// TwinCAT 3 PLC project Untitled1
// ProgramVersion: 3.1.4024.0
// libraries:
//   Tc2_Standard, * (Beckhoff Automation GmbH)
//   Tc2_System, * (Beckhoff Automation GmbH)
//   Tc2_Utilities, * (Beckhoff Automation GmbH)
//   Tc3_Module, * (Beckhoff Automation GmbH)
// project tree:
//   / PlcTask.TcTTO
//   Lib/Any/ ToAnyType.TcPOU (not stored)
//   Lib/ MAIN.TcPOU (not stored)
//   Lib/PrimitiveValues/ ValueLrealRead.TcPOU (not stored), ValueLreal.TcPOU, ValueByte.TcPOU (not stored), ValueByteRead.TcPOU (not stored), ValueDate.TcPOU (not stored), ValueDateRead.TcPOU, ValueDint.TcPOU (not stored), ValueDintRead.TcPOU (not stored), ValueDt.TcPOU (not stored), ValueDtRead.TcPOU (not stored), ValueDword.TcPOU (not stored), ValueDwordRead.TcPOU (not stored), ValueInt.TcPOU, ValueIntRead.TcPOU (not stored), ValueLint.TcPOU, ValueLintRead.TcPOU, ValueLtime.TcPOU (not stored), ValueLtimeRead.TcPOU, ValueLword.TcPOU (not stored), ValueLwordRead.TcPOU (not stored), ValueReal.TcPOU (not stored), ValueRealRead.TcPOU, ValueSint.TcPOU (not stored), ValueSintRead.TcPOU, ValueString.TcPOU, ValueStringRead.TcPOU (not stored), ValueTime.TcPOU (not stored), ValueTimeRead.TcPOU (not stored), ValueTod.TcPOU, ValueTodRead.TcPOU (not stored), ValueUdint.TcPOU (not stored), ValueUdintRead.TcPOU, ValueUint.TcPOU (not stored), ValueUintRead.TcPOU (not stored), ValueUlint.TcPOU, ValueUlintRead.TcPOU, ValueUsint.TcPOU (not stored), ValueUsintRead.TcPOU (not stored), ValueWord.TcPOU (not stored), ValueWordRead.TcPOU (not stored), ValueWstring.TcPOU, ValueWstringRead.TcPOU (not stored)
//   Lib/Startable/ CommandStatus.TcIO (not stored), Startable.TcIO
//   Lib/Value/ Value.TcIO, ValueBase.TcPOU, ValueWithType.TcIO, ValueRead.TcIO (not stored), ValueType.TcDUT
//   Lib/Conversion/ ConvertAnyType.TcPOU (not stored)
// real-time tasks:
//   TASK PlcTask: cycle T#10ms, priority 20, ADS port 350

CONFIGURATION Untitled1
    RESOURCE PLC ON TwinCAT3
        TASK PlcTask(INTERVAL := T#10ms, PRIORITY := 20);
        PROGRAM MAIN WITH PlcTask : MAIN;
    END_RESOURCE
END_CONFIGURATION

// ---- Lib/Value/ValueType.TcDUT
TYPE ValueType : __SYSTEM.TYPE_CLASS; END_TYPE

// ---- Lib/Startable/Startable.TcIO
{attribute 'linkalways'}
INTERFACE Startable EXTENDS __SYSTEM.IQueryInterface

METHOD Start : CommandStatus
END_METHOD

END_INTERFACE

// ---- Lib/Value/Value.TcIO
{attribute 'linkalways'}
INTERFACE Value EXTENDS ValueRead

METHOD Set : BOOL
VAR_INPUT
	source : ANY;
END_VAR
END_METHOD

METHOD SetFromString : BOOL
VAR_INPUT
	value : T_MaxString;
END_VAR
END_METHOD

METHOD SetFromType : BOOL
VAR_INPUT
	source : __SYSTEM.AnyType;
END_VAR
END_METHOD

END_INTERFACE

// ---- Lib/Value/ValueWithType.TcIO
INTERFACE ValueWithType EXTENDS __SYSTEM.IQueryInterface

{attribute 'monitoring' := 'call'}
PROPERTY ValueType : ValueType
GET
END_GET
END_PROPERTY

END_INTERFACE

// ---- Lib/PrimitiveValues/ValueLreal.TcPOU
{attribute 'linkalways'}
{attribute 'hide_all_locals'}
FUNCTION_BLOCK ValueLreal EXTENDS ValueLrealRead IMPLEMENTS Value
VAR
END_VAR

METHOD Set : BOOL
VAR_INPUT
	source : ANY;
END_VAR
Set := ConvertAnyType(source, thisAnyType);
END_METHOD

METHOD SetFromString : BOOL
VAR_INPUT
	value : T_MaxString;
END_VAR
thisValue := STRING_TO_LREAL(value);

SetFromString := TRUE;
END_METHOD

METHOD SetFromType : BOOL
VAR_INPUT
	source : __SYSTEM.AnyType;
END_VAR
SetFromType := ConvertAnyType(source, thisAnyType);
END_METHOD

END_FUNCTION_BLOCK

// ---- Lib/Value/ValueBase.TcPOU
{attribute 'linkalways'}
{attribute 'hide_all_locals'}
FUNCTION_BLOCK ABSTRACT ValueBase IMPLEMENTS ValueWithType
VAR
	_ValueType : ValueType;
	thisAnyType : __SYSTEM.AnyType;
END_VAR

{attribute 'call_after_global_init_slot' := '1'}
{attribute 'call_after_online_change_slot' := '1'}
METHOD PROTECTED ABSTRACT GetThisAnyType
VAR_INPUT
END_VAR
END_METHOD

{attribute 'monitoring' := 'call'}
PROPERTY ValueType : ValueType
GET
ValueType := _ValueType;
END_GET
END_PROPERTY

END_FUNCTION_BLOCK

// ---- Lib/PrimitiveValues/ValueDateRead.TcPOU
{attribute 'linkalways'}
{attribute 'hide_all_locals'}
FUNCTION_BLOCK ValueDateRead EXTENDS ValueBase IMPLEMENTS ValueRead
VAR
	thisValue : DATE;
END_VAR

{attribute 'call_after_global_init_slot' := '1'}
{attribute 'call_after_online_change_slot' := '1'}
METHOD PROTECTED GetThisAnyType
VAR_INPUT
END_VAR
thisAnyType := ToAnyType(thisValue);
END_METHOD

METHOD GetAsType : BOOL
VAR_INPUT
	destination : __SYSTEM.AnyType;
END_VAR
GetAsType := ConvertAnyType(thisAnyType, destination);
END_METHOD

METHOD GetAsString : T_MaxString
VAR_INPUT
END_VAR
GetAsString := DATE_TO_STRING(thisValue);
END_METHOD

METHOD Get : BOOL
VAR_INPUT
	destination : ANY;
END_VAR
Get := ConvertAnyType(thisAnyType, destination);
END_METHOD

METHOD FB_init : BOOL
VAR_INPUT
	bInitRetains : BOOL; // if TRUE, the retain variables are initialized (warm start / cold start)
	bInCopyCode : BOOL;  // if TRUE, the instance afterwards gets moved into the copy code (online change)
END_VAR
_ValueType := __SYSTEM.TYPE_CLASS.TYPE_DATE;
END_METHOD

{attribute 'monitoring' := 'call'}
PROPERTY Value : DATE
GET
Value := thisValue;
END_GET
END_PROPERTY

END_FUNCTION_BLOCK

// ---- Lib/PrimitiveValues/ValueInt.TcPOU
{attribute 'linkalways'}
{attribute 'hide_all_locals'}
FUNCTION_BLOCK ValueInt EXTENDS ValueIntRead IMPLEMENTS Value
VAR
END_VAR

METHOD SetFromType : BOOL
VAR_INPUT
	source : __SYSTEM.AnyType;
END_VAR
SetFromType := ConvertAnyType(source, thisAnyType);
END_METHOD

METHOD SetFromString : BOOL
VAR_INPUT
	value : T_MaxString;
END_VAR
thisValue := STRING_TO_INT(value);

SetFromString := TRUE;
END_METHOD

METHOD Set : BOOL
VAR_INPUT
	source : ANY;
END_VAR
Set := ConvertAnyType(source, thisAnyType);
END_METHOD

END_FUNCTION_BLOCK

// ---- Lib/PrimitiveValues/ValueLint.TcPOU
{attribute 'linkalways'}
{attribute 'hide_all_locals'}
FUNCTION_BLOCK ValueLint EXTENDS ValueLintRead IMPLEMENTS Value
VAR
END_VAR

METHOD SetFromType : BOOL
VAR_INPUT
	source : __SYSTEM.AnyType;
END_VAR
SetFromType := ConvertAnyType(source, thisAnyType);
END_METHOD

METHOD SetFromString : BOOL
VAR_INPUT
	value : T_MaxString;
END_VAR
thisValue := STRING_TO_LINT(value);

SetFromString := TRUE;
END_METHOD

METHOD Set : BOOL
VAR_INPUT
	source : ANY;
END_VAR
Set := ConvertAnyType(source, thisAnyType);
END_METHOD

END_FUNCTION_BLOCK

// ---- Lib/PrimitiveValues/ValueLintRead.TcPOU
{attribute 'linkalways'}
{attribute 'hide_all_locals'}
FUNCTION_BLOCK ValueLintRead EXTENDS ValueBase IMPLEMENTS ValueRead
VAR
	thisValue : LINT;
END_VAR

{attribute 'call_after_global_init_slot' := '1'}
{attribute 'call_after_online_change_slot' := '1'}
METHOD PROTECTED GetThisAnyType
VAR_INPUT
END_VAR
thisAnyType := ToAnyType(thisValue);
END_METHOD

METHOD GetAsType : BOOL
VAR_INPUT
	destination : __SYSTEM.AnyType;
END_VAR
GetAsType := ConvertAnyType(thisAnyType, destination);
END_METHOD

METHOD GetAsString : T_MaxString
VAR_INPUT
END_VAR
GetAsString := TO_STRING(thisValue);
END_METHOD

METHOD Get : BOOL
VAR_INPUT
	destination : ANY;
END_VAR
Get := ConvertAnyType(thisAnyType, destination);
END_METHOD

METHOD FB_init : BOOL
VAR_INPUT
	bInitRetains : BOOL; // if TRUE, the retain variables are initialized (warm start / cold start)
	bInCopyCode : BOOL;  // if TRUE, the instance afterwards gets moved into the copy code (online change)
END_VAR
_ValueType := __SYSTEM.TYPE_CLASS.TYPE_LINT;
END_METHOD

{attribute 'monitoring' := 'call'}
PROPERTY Value : LINT
GET
Value := thisValue;
END_GET
END_PROPERTY

END_FUNCTION_BLOCK

// ---- Lib/PrimitiveValues/ValueLtimeRead.TcPOU
{attribute 'linkalways'}
{attribute 'hide_all_locals'}
FUNCTION_BLOCK ValueLtimeRead EXTENDS ValueBase IMPLEMENTS ValueRead
VAR
	thisValue : LTIME;
END_VAR

{attribute 'call_after_global_init_slot' := '1'}
{attribute 'call_after_online_change_slot' := '1'}
METHOD PROTECTED GetThisAnyType
VAR_INPUT
END_VAR
thisAnyType := ToAnyType(thisValue);
END_METHOD

METHOD GetAsType : BOOL
VAR_INPUT
	destination : __SYSTEM.AnyType;
END_VAR
GetAsType := ConvertAnyType(thisAnyType, destination);
END_METHOD

METHOD GetAsString : T_MaxString
VAR_INPUT
END_VAR
GetAsString := LTIME_TO_STRING(thisValue);
END_METHOD

METHOD Get : BOOL
VAR_INPUT
	destination : ANY;
END_VAR
Get := ConvertAnyType(thisAnyType, destination);
END_METHOD

METHOD FB_init : BOOL
VAR_INPUT
	bInitRetains : BOOL; // if TRUE, the retain variables are initialized (warm start / cold start)
	bInCopyCode : BOOL;  // if TRUE, the instance afterwards gets moved into the copy code (online change)
END_VAR
_ValueType := __SYSTEM.TYPE_CLASS.TYPE_LTIME;
END_METHOD

{attribute 'monitoring' := 'call'}
PROPERTY Value : LTIME
GET
Value := thisValue;
END_GET
END_PROPERTY

END_FUNCTION_BLOCK

// ---- Lib/PrimitiveValues/ValueRealRead.TcPOU
{attribute 'linkalways'}
{attribute 'hide_all_locals'}
FUNCTION_BLOCK ValueRealRead EXTENDS ValueBase IMPLEMENTS ValueRead
VAR
	thisValue : REAL;
END_VAR

{attribute 'call_after_global_init_slot' := '1'}
{attribute 'call_after_online_change_slot' := '1'}
METHOD PROTECTED GetThisAnyType
VAR_INPUT
END_VAR
thisAnyType := ToAnyType(thisValue);
END_METHOD

METHOD GetAsType : BOOL
VAR_INPUT
	destination : __SYSTEM.AnyType;
END_VAR
GetAsType := ConvertAnyType(thisAnyType, destination);
END_METHOD

METHOD GetAsString : T_MaxString
VAR_INPUT
END_VAR
GetAsString := TO_STRING(thisValue);
END_METHOD

METHOD Get : BOOL
VAR_INPUT
	destination : ANY;
END_VAR
Get := ConvertAnyType(thisAnyType, destination);
END_METHOD

METHOD FB_init : BOOL
VAR_INPUT
	bInitRetains : BOOL; // if TRUE, the retain variables are initialized (warm start / cold start)
	bInCopyCode : BOOL;  // if TRUE, the instance afterwards gets moved into the copy code (online change)
END_VAR
_ValueType := __SYSTEM.TYPE_CLASS.TYPE_REAL;
END_METHOD

{attribute 'monitoring' := 'call'}
PROPERTY Value : REAL
GET
Value := thisValue;
END_GET
END_PROPERTY

END_FUNCTION_BLOCK

// ---- Lib/PrimitiveValues/ValueSintRead.TcPOU
{attribute 'linkalways'}
{attribute 'hide_all_locals'}
FUNCTION_BLOCK ValueSintRead EXTENDS ValueBase IMPLEMENTS ValueRead
VAR
	thisValue : SINT;
END_VAR

{attribute 'call_after_global_init_slot' := '1'}
{attribute 'call_after_online_change_slot' := '1'}
METHOD PROTECTED GetThisAnyType
VAR_INPUT
END_VAR
thisAnyType := ToAnyType(thisValue);
END_METHOD

METHOD GetAsType : BOOL
VAR_INPUT
	destination : __SYSTEM.AnyType;
END_VAR
GetAsType := ConvertAnyType(thisAnyType, destination);
END_METHOD

METHOD GetAsString : T_MaxString
VAR_INPUT
END_VAR
GetAsString := TO_STRING(thisValue);
END_METHOD

METHOD Get : BOOL
VAR_INPUT
	destination : ANY;
END_VAR
Get := ConvertAnyType(thisAnyType, destination);
END_METHOD

METHOD FB_init : BOOL
VAR_INPUT
	bInitRetains : BOOL; // if TRUE, the retain variables are initialized (warm start / cold start)
	bInCopyCode : BOOL;  // if TRUE, the instance afterwards gets moved into the copy code (online change)
END_VAR
_ValueType := __SYSTEM.TYPE_CLASS.TYPE_SINT;
END_METHOD

{attribute 'monitoring' := 'call'}
PROPERTY Value : SINT
GET
Value := thisValue;
END_GET
END_PROPERTY

END_FUNCTION_BLOCK

// ---- Lib/PrimitiveValues/ValueString.TcPOU
{attribute 'linkalways'}
{attribute 'hide_all_locals'}
FUNCTION_BLOCK ValueString EXTENDS ValueStringRead IMPLEMENTS Value
VAR
END_VAR

METHOD SetFromType : BOOL
VAR_INPUT
	source : __SYSTEM.AnyType;
END_VAR
SetFromType := ConvertAnyType(source, thisAnyType);
END_METHOD

METHOD SetFromString : BOOL
VAR_INPUT
	value : T_MaxString;
END_VAR
thisValue := value;

SetFromString := TRUE;
END_METHOD

METHOD Set : BOOL
VAR_INPUT
	source : ANY;
END_VAR
Set := ConvertAnyType(source, thisAnyType);
END_METHOD

END_FUNCTION_BLOCK

// ---- Lib/PrimitiveValues/ValueTod.TcPOU
{attribute 'linkalways'}
{attribute 'hide_all_locals'}
FUNCTION_BLOCK ValueTod EXTENDS ValueTodRead IMPLEMENTS Value
VAR
END_VAR

METHOD SetFromType : BOOL
VAR_INPUT
	source : __SYSTEM.AnyType;
END_VAR
SetFromType := ConvertAnyType(source, thisAnyType);
END_METHOD

METHOD SetFromString : BOOL
VAR_INPUT
	value : T_MaxString;
END_VAR
thisValue := STRING_TO_TOD(value);

SetFromString := TRUE;
END_METHOD

METHOD Set : BOOL
VAR_INPUT
	source : ANY;
END_VAR
Set := ConvertAnyType(source, thisAnyType);
END_METHOD

END_FUNCTION_BLOCK

// ---- Lib/PrimitiveValues/ValueUdintRead.TcPOU
{attribute 'linkalways'}
{attribute 'hide_all_locals'}
FUNCTION_BLOCK ValueUdintRead EXTENDS ValueBase IMPLEMENTS ValueRead
VAR
	thisValue : UDINT;
END_VAR

{attribute 'call_after_global_init_slot' := '1'}
{attribute 'call_after_online_change_slot' := '1'}
METHOD PROTECTED GetThisAnyType
VAR_INPUT
END_VAR
thisAnyType := ToAnyType(thisValue);
END_METHOD

METHOD GetAsType : BOOL
VAR_INPUT
	destination : __SYSTEM.AnyType;
END_VAR
GetAsType := ConvertAnyType(thisAnyType, destination);
END_METHOD

METHOD GetAsString : T_MaxString
VAR_INPUT
END_VAR
GetAsString := TO_STRING(thisValue);
END_METHOD

METHOD Get : BOOL
VAR_INPUT
	destination : ANY;
END_VAR
Get := ConvertAnyType(thisAnyType, destination);
END_METHOD

METHOD FB_init : BOOL
VAR_INPUT
	bInitRetains : BOOL; // if TRUE, the retain variables are initialized (warm start / cold start)
	bInCopyCode : BOOL;  // if TRUE, the instance afterwards gets moved into the copy code (online change)
END_VAR
_ValueType := __SYSTEM.TYPE_CLASS.TYPE_UDINT;
END_METHOD

{attribute 'monitoring' := 'call'}
PROPERTY Value : UDINT
GET
Value := thisValue;
END_GET
END_PROPERTY

END_FUNCTION_BLOCK

// ---- Lib/PrimitiveValues/ValueUlint.TcPOU
{attribute 'linkalways'}
{attribute 'hide_all_locals'}
FUNCTION_BLOCK ValueUlint EXTENDS ValueUlintRead IMPLEMENTS Value
VAR
END_VAR

METHOD SetFromType : BOOL
VAR_INPUT
	source : __SYSTEM.AnyType;
END_VAR
SetFromType := ConvertAnyType(source, thisAnyType);
END_METHOD

METHOD SetFromString : BOOL
VAR_INPUT
	value : T_MaxString;
END_VAR
thisValue := STRING_TO_ULINT(value);

SetFromString := TRUE;
END_METHOD

METHOD Set : BOOL
VAR_INPUT
	source : ANY;
END_VAR
Set := ConvertAnyType(source, thisAnyType);
END_METHOD

END_FUNCTION_BLOCK

// ---- Lib/PrimitiveValues/ValueUlintRead.TcPOU
{attribute 'linkalways'}
{attribute 'hide_all_locals'}
FUNCTION_BLOCK ValueUlintRead EXTENDS ValueBase IMPLEMENTS ValueRead
VAR
	thisValue : ULINT;
END_VAR

{attribute 'call_after_global_init_slot' := '1'}
{attribute 'call_after_online_change_slot' := '1'}
METHOD PROTECTED GetThisAnyType
VAR_INPUT
END_VAR
thisAnyType := ToAnyType(thisValue);
END_METHOD

METHOD GetAsType : BOOL
VAR_INPUT
	destination : __SYSTEM.AnyType;
END_VAR
GetAsType := ConvertAnyType(thisAnyType, destination);
END_METHOD

METHOD GetAsString : T_MaxString
VAR_INPUT
END_VAR
GetAsString := TO_STRING(thisValue);
END_METHOD

METHOD Get : BOOL
VAR_INPUT
	destination : ANY;
END_VAR
Get := ConvertAnyType(thisAnyType, destination);
END_METHOD

METHOD FB_init : BOOL
VAR_INPUT
	bInitRetains : BOOL; // if TRUE, the retain variables are initialized (warm start / cold start)
	bInCopyCode : BOOL;  // if TRUE, the instance afterwards gets moved into the copy code (online change)
END_VAR
_ValueType := __SYSTEM.TYPE_CLASS.TYPE_ULINT;
END_METHOD

{attribute 'monitoring' := 'call'}
PROPERTY Value : ULINT
GET
Value := thisValue;
END_GET
END_PROPERTY

END_FUNCTION_BLOCK

// ---- Lib/PrimitiveValues/ValueWstring.TcPOU
{attribute 'linkalways'}
{attribute 'hide_all_locals'}
FUNCTION_BLOCK ValueWstring EXTENDS ValueWstringRead IMPLEMENTS Value
VAR
END_VAR

METHOD SetFromType : BOOL
VAR_INPUT
	source : __SYSTEM.AnyType;
END_VAR
SetFromType := ConvertAnyType(source, thisAnyType);
END_METHOD

METHOD SetFromString : BOOL
VAR_INPUT
	value : T_MaxString;
END_VAR
thisValue := STRING_TO_WSTRING(value);

SetFromString := TRUE;
END_METHOD

METHOD Set : BOOL
VAR_INPUT
	source : ANY;
END_VAR
Set := ConvertAnyType(source, thisAnyType);
END_METHOD

END_FUNCTION_BLOCK
